Fanuc KAREL source: ka00119.KL

PROGRAM KA00119
%STACKSIZE=65535
%PRIORITY=65535
%NOLOCKGROUP
VAR
DST : ARRAY[2] OF BYTE
-- UNRESOLVED DECLARATIONS (source type spelling not recovered)
-- SRC : TYPE_0x001C (type_u16=0x001C)
BEGIN
-- UNRESOLVED_PC line 7 opcodes [9D 22 A5] marker_code=0
-- UNRESOLVED_PC line 8 opcodes [21 22 9D 33 B2] marker_code=15
END KA00119
